{attribute 'qualified_only'}
VAR_GLOBAL
END_VAR

(* stored: Version 1.1.0.1, ProductVersion 3.1.4022.7
   GVL GVL_05_Manual_Step_Motor_BOX_X: Id {4d2e7aea-8582-4eb6-90a1-cdb6dd599e56} *)
